// TIA Portal V20 export
TYPE "Analog_Ctrl_DT"
   STRUCT
      Type_of_probe { ExternalVisible := 'False'} : Int;   // PT100=0, PT1000=1, NTC=2, RES600=3, 0-10V=4, -10+10V=5, 0-2000=6 / PT100=0(FC71:0, PT1000=1(FC71:1), NTC=2(FC74), RES600=3
      Target_value : Real;
      SWRealValue { ExternalVisible := 'False'} : Real;
      HWWordValue : Word;
      Time_delay { ExternalVisible := 'False'} : Time;
      Threshold_Alarm_min { ExternalVisible := 'False'} : Real;
      Threshold_Warning_min { ExternalVisible := 'False'} : Real;
      Threshold_Warning_max { ExternalVisible := 'False'} : Real;
      Threshold_Alarm_max { ExternalVisible := 'False'} : Real;
      Num_alarm_min { ExternalVisible := 'False'} : Int := -1;
      Num_warning_min { ExternalVisible := 'False'} : Int := -1;
      Num_warning_max { ExternalVisible := 'False'} : Int := -1;
      Num_alarm_max { ExternalVisible := 'False'} : Int := -1;
      Num_alarm_out_of_range { ExternalVisible := 'False'} : Int := -1;
      Stop_machine { ExternalVisible := 'False'} : Bool;
      Bad_part_on_laser { ExternalVisible := 'False'} : Bool;
      axFactor : Real;
      bOffset : Real;
      iLimitUp : Real;
      iLimitDown : Real;
   END_STRUCT;
END_TYPE
